PROGRAM MAIN
VAR
	ConveyorControl : BOOL;
	Timeout : TOF;
END_VAR

IF NOT GVL.StopButton OR NOT GVL.EmergencyStopButton THEN
	
	ConveyorControl := FALSE;
	
ELSIF GVL.StartButton AND GVL.StopButton AND GVL.EmergencyStopButton THEN
	
	ConveyorControl := TRUE;
	
END_IF

Timeout(IN:= ConveyorControl AND GVL.ProductDetectedSensor, PT := T#5S);

GVL.MotorContactor := ConveyorControl AND Timeout.Q AND NOT GVL.ConveyorFullSensor;

END_PROGRAM

(* stored: Version 1.1.0.1, ProductVersion 3.1.4024.11
   POU MAIN: Id {bb1f3822-6112-4b9b-955d-290fdd8d76c0}, SpecialFunc None *)
